// TIA Portal project "PLC_Leonardo_2022_10_27_Rev01" (V16)

(* hardware
DEVICE "S7-1200 station_1"  S7-1200 Station
   slot 0: "Telaio di montaggio_0"  S7-1200 Rack  Rack  V1.0
   slot 1: "PLC_1"  CPU 1212C DC/DC/DC  6ES7 212-1AE40-0XB0  V4.4
*)

// ===== PLC "PLC_1"  CPU 1212C DC/DC/DC =====

DATA_BLOCK "Scabio_DB"   // DB1
{ S7_Optimized_Access := 'FALSE' }
VERSION : 0.1
   VAR
      Cucina : Struct
         SNS_C1_Seduto_Al_Tavolo : Bool;
         SNS_C2_Presenza_Nella_Stanza : Bool;
         SNS_C3_Piatti_Sul_Tavolo : Bool;
         SNS_C4_Chiusura_Frigor : Bool;
         SNS_C5 : Bool;
         SNS_C6 : Bool;
         SNS_C7 : Bool;
         SNS_C8 : Bool;
         SNS_C9 : Bool;
         SNS_C10 : Bool;
         SNS_C11 : Bool;
         SNS_C12 : Bool;
         SNS_C13 : Bool;
         SNS_C14 : Bool;
         SNS_C15 : Bool;
         SNS_C16 : Bool;
      END_STRUCT;
      Camera : Struct
         SNS_B1_Sdraiato_Sul_Letto : Bool;
         SNS_B2_Presenza_Nella_Stanza : Bool;
         SNS_B3 : Bool;
         SNS_B4 : Bool;
         SNS_B5 : Bool;
         SNS_B6 : Bool;
         SNS_B7 : Bool;
         SNS_B8 : Bool;
         SNS_B9 : Bool;
         SNS_B10 : Bool;
         SNS_B11 : Bool;
         SNS_B12 : Bool;
         SNS_B13 : Bool;
         SNS_B14 : Bool;
         SNS_B15 : Bool;
         SNS_B16 : Bool;
      END_STRUCT;
      Sala : Struct
         SNS_S1_Presenza_Sul_Divano : Bool;
         SNS_S2_Presenza_Nella_Stanza : Bool;
         SNS_S3 : Bool;
         SNS_S4 : Bool;
         SNS_S5_Passaggio_Camera_Inferiore : Bool;
         SNS_S6 : Bool;
         SNS_S7 : Bool;
         SNS_S8 : Bool;
         SNS_S9 : Bool;
         SNS_S10 : Bool;
         SNS_S11 : Bool;
         SNS_S12 : Bool;
         SNS_S13 : Bool;
         SNS_S14 : Bool;
         SNS_S15 : Bool;
         SNS_S16 : Bool;
      END_STRUCT;
   END_VAR
BEGIN
END_DATA_BLOCK

ORGANIZATION_BLOCK "Main"   // OB1, LAD, ProgramCycle
TITLE = "Main Program Sweep (Cycle)"
{ S7_Optimized_Access := 'TRUE' }
VERSION : 0.1
   VAR_INPUT
      Initial_Call : Bool;   // Initial call of this OB
      Remanence : Bool;   // =True, if remanent data are available
   END_VAR
BEGIN
END_ORGANIZATION_BLOCK